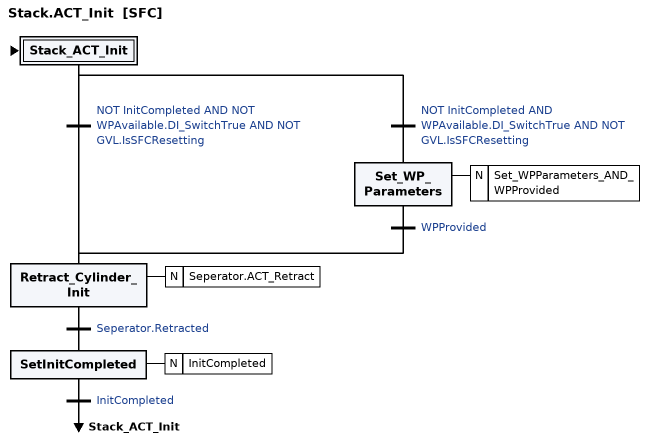
INITIAL_STEP Stack_ACT_Init:
END_STEP
TRANSITION FROM Stack_ACT_Init TO Retract_Cylinder_Init
  := NOT InitCompleted AND NOT WPAvailable.DI_SwitchTrue AND NOT
                                                    GVL.IsSFCResetting;
END_TRANSITION
TRANSITION FROM Stack_ACT_Init TO Set_WP_Parameters
  := NOT InitCompleted AND WPAvailable.DI_SwitchTrue AND NOT
                                                    GVL.IsSFCResetting;
END_TRANSITION
STEP Set_WP_Parameters:
  Set_WPParameters_AND_WPProvided(N);
END_STEP
TRANSITION FROM Set_WP_Parameters TO Retract_Cylinder_Init
  := WPProvided;
END_TRANSITION
STEP Retract_Cylinder_Init:
  Seperator.ACT_Retract(N);
END_STEP
TRANSITION FROM Retract_Cylinder_Init TO SetInitCompleted
  := Seperator.Retracted;
END_TRANSITION
STEP SetInitCompleted:
  InitCompleted(N);
END_STEP
TRANSITION FROM SetInitCompleted TO Stack_ACT_Init
  := InitCompleted;
END_TRANSITION
END_ACTION
END_FUNCTION_BLOCK

FUNCTION_BLOCK Stamp
                                            VAR_INPUT
                                            //Hardware
                                            Panel : OperationPanel;
                                            PressureSensor : PressureSensor;
                                            PropValve : ProportionalValve;
                                            WPAvailable : MicroSwitch;
                                            StampingCylinder : MonostableCylinder;
                                            SlidingCylinder : BistableCylinder;

                                            //Software
                                            StartButton : BOOL;
                                            InitCompleted : BOOL;
                                            AutomaticExecuteCompleted : BOOL;
                                            EmergencyStop : BOOL;
                                            SoftwareEmergency : BOOL;
                                            EmergencyHandled : BOOL;
                                            SFCReset : BOOL; //Only for SFC implementation
                                            END_VAR
                                            VAR_OUTPUT
                                            //Software
                                            IsStamping : BOOL;
                                            WPStamped : BOOL;
                                            WPType_White : BOOL;
                                            WPType_Black : BOOL;
                                            WPType_Metallic : BOOL;
                                            END_VAR
                                            VAR
                                            //Software
                                            Timer : TON;
                                            Check_Allowed_To_Operate : BOOL;
                                            Check_WPType_White : BOOL;
                                            Check_WPType_Black : BOOL;
                                            Check_WPType_Metallic : BOOL;
                                            Check_Stamp_WPAvailable : BOOL;
                                            END_VAR

                                    Panel();
                                        StartButton := Panel.StartButton;
                                        EmergencyStop := Panel.EmergencyStop;
                                        Check_Allowed_To_Operate := Main.Crane_Allow_Stamp_to_Operate;
                                        Check_WPType_White:=Main.Crane_WPType_White;
                                        Check_WPType_Black:=Main.Crane_WPType_Black;
                                        Check_WPType_Metallic:=Main.Crane_WPType_Metallic;
                                        Check_Stamp_WPAvailable:=Main.Stamp_WPAvailable;
                                    
                                

ACTION ExtendStampingCylinder_AND_Timer1500ms:
                                            StampingCylinder.ACT_Extend();
                                                Timer(IN:=TRUE, PT:=T#1500MS);
                                            
                                        
END_ACTION

ACTION Reset_Pressure:
                                            PropValve.AO_SetPressure:=0;
                                            
                                        
END_ACTION

ACTION Reset_Timer:
                                            Timer(IN:=FALSE);
                                        
END_ACTION

ACTION Reset_Variables:
                                            InitCompleted := FALSE;
                                                AutomaticExecuteCompleted := FALSE;

                                                propValve.AO_SetPressure:=0;
                                                IsStamping:=FALSE;
                                                WPStamped:=FALSE;
                                                WPType_Black := FALSE;
                                                WPType_White := FALSE;
                                                WPType_Metallic := FALSE;
                                            
                                        
END_ACTION

ACTION Set_HeavyPressure:
                                            
                                                PropValve.AO_SetPressure:=7000;
                                            
                                        
END_ACTION

ACTION Set_LightPressure:
                                            
                                                PropValve.AO_SetPressure:=4000;
                                            
                                        
END_ACTION

ACTION Set_Timer1000ms:
                                            Timer(IN:=TRUE, PT:=T#1000MS);
                                            
                                        
END_ACTION

ACTION Set_Timer500ms:
                                            Timer(IN:=TRUE, PT:=T#500ms);
                                            
                                        
END_ACTION

ACTION Set_WPType:
                                            WPType_White :=
                                                Check_WPType_White;
                                                WPType_Black := Check_WPType_Black;
                                                WPType_Metallic := Check_WPType_Metallic;
                                            
                                        
END_ACTION

ACTION ACT_Stamp:
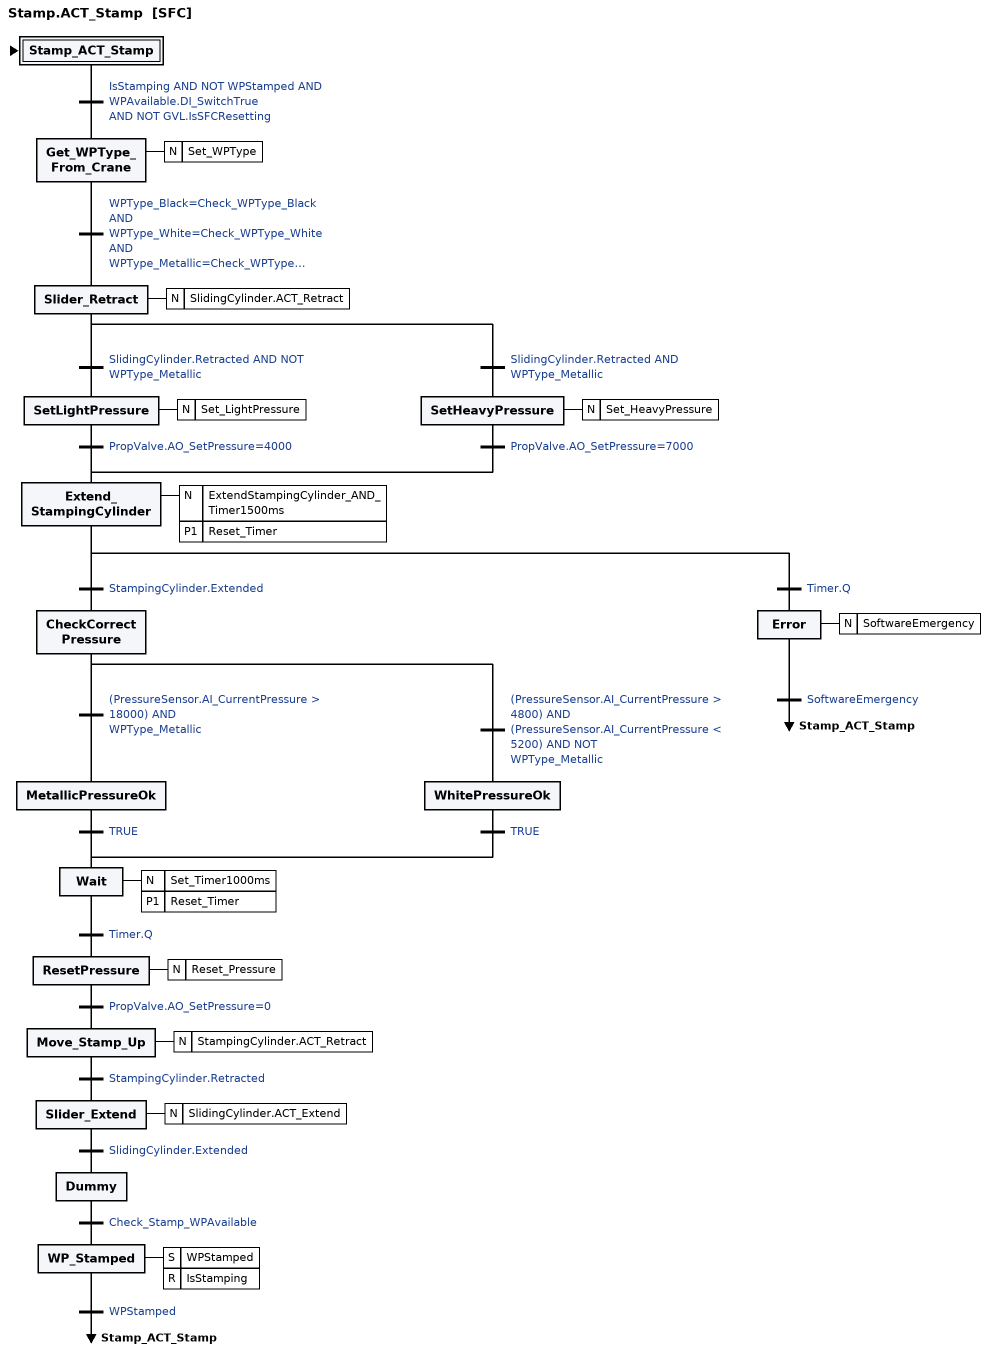
INITIAL_STEP Stamp_ACT_Stamp:
END_STEP
TRANSITION FROM Stamp_ACT_Stamp TO Get_WPType_From_Crane
  := IsStamping AND NOT WPStamped AND WPAvailable.DI_SwitchTrue
                                                    AND NOT GVL.IsSFCResetting;
END_TRANSITION
STEP Get_WPType_From_Crane:
  Set_WPType(N);
END_STEP
TRANSITION FROM Get_WPType_From_Crane TO Slider_Retract
  := WPType_Black=Check_WPType_Black AND
                                                    WPType_White=Check_WPType_White AND
                                                    WPType_Metallic=Check_WPType_Metallic;
END_TRANSITION
STEP Slider_Retract:
  SlidingCylinder.ACT_Retract(N);
END_STEP
TRANSITION FROM Slider_Retract TO SetLightPressure
  := SlidingCylinder.Retracted AND NOT WPType_Metallic;
END_TRANSITION
TRANSITION FROM Slider_Retract TO SetHeavyPressure
  := SlidingCylinder.Retracted AND WPType_Metallic;
END_TRANSITION
STEP SetLightPressure:
  Set_LightPressure(N);
END_STEP
TRANSITION FROM SetLightPressure TO Extend_StampingCylinder
  := PropValve.AO_SetPressure=4000;
END_TRANSITION
STEP SetHeavyPressure:
  Set_HeavyPressure(N);
END_STEP
TRANSITION FROM SetHeavyPressure TO Extend_StampingCylinder
  := PropValve.AO_SetPressure=7000;
END_TRANSITION
STEP Extend_StampingCylinder:
  ExtendStampingCylinder_AND_Timer1500ms(N);
  Reset_Timer(P1);
END_STEP
TRANSITION FROM Extend_StampingCylinder TO CheckCorrectPressure
  := StampingCylinder.Extended;
END_TRANSITION
TRANSITION FROM Extend_StampingCylinder TO Error
  := Timer.Q;
END_TRANSITION
STEP CheckCorrectPressure:
END_STEP
TRANSITION FROM CheckCorrectPressure TO MetallicPressureOk
  := (PressureSensor.AI_CurrentPressure > 18000) AND
                                                    WPType_Metallic;
END_TRANSITION
TRANSITION FROM CheckCorrectPressure TO WhitePressureOk
  := (PressureSensor.AI_CurrentPressure > 4800) AND
                                                    (PressureSensor.AI_CurrentPressure < 5200) AND NOT
                                                    WPType_Metallic;
END_TRANSITION
STEP MetallicPressureOk:
END_STEP
TRANSITION FROM MetallicPressureOk TO Wait
  := TRUE;
END_TRANSITION
STEP WhitePressureOk:
END_STEP
TRANSITION FROM WhitePressureOk TO Wait
  := TRUE;
END_TRANSITION
STEP Error:
  SoftwareEmergency(N);
END_STEP
TRANSITION FROM Error TO Stamp_ACT_Stamp
  := SoftwareEmergency;
END_TRANSITION
STEP Wait:
  Set_Timer1000ms(N);
  Reset_Timer(P1);
END_STEP
TRANSITION FROM Wait TO ResetPressure
  := Timer.Q;
END_TRANSITION
STEP ResetPressure:
  Reset_Pressure(N);
END_STEP
TRANSITION FROM ResetPressure TO Move_Stamp_Up
  := PropValve.AO_SetPressure=0;
END_TRANSITION
STEP Move_Stamp_Up:
  StampingCylinder.ACT_Retract(N);
END_STEP
TRANSITION FROM Move_Stamp_Up TO Slider_Extend
  := StampingCylinder.Retracted;
END_TRANSITION
STEP Slider_Extend:
  SlidingCylinder.ACT_Extend(N);
END_STEP
TRANSITION FROM Slider_Extend TO Dummy
  := SlidingCylinder.Extended;
END_TRANSITION
STEP Dummy:
END_STEP
TRANSITION FROM Dummy TO WP_Stamped
  := Check_Stamp_WPAvailable;
END_TRANSITION
STEP WP_Stamped:
  WPStamped(S);
  IsStamping(R);
END_STEP
TRANSITION FROM WP_Stamped TO Stamp_ACT_Stamp
  := WPStamped;
END_TRANSITION
END_ACTION

ACTION ACT_AutomaticExecute:
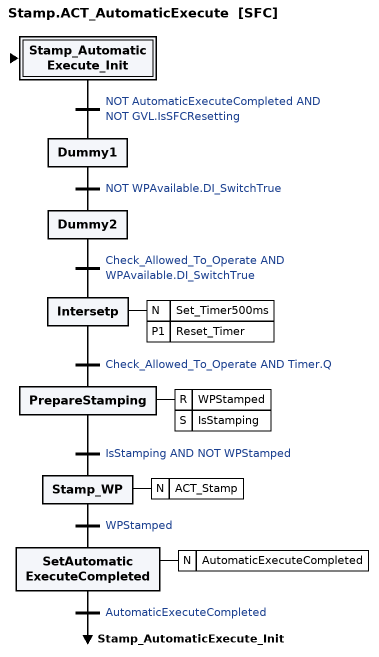
INITIAL_STEP Stamp_AutomaticExecute_Init:
END_STEP
TRANSITION FROM Stamp_AutomaticExecute_Init TO Dummy1
  := NOT AutomaticExecuteCompleted AND NOT GVL.IsSFCResetting;
END_TRANSITION
STEP Dummy1:
END_STEP
TRANSITION FROM Dummy1 TO Dummy2
  := NOT WPAvailable.DI_SwitchTrue;
END_TRANSITION
STEP Dummy2:
END_STEP
TRANSITION FROM Dummy2 TO Intersetp
  := Check_Allowed_To_Operate AND WPAvailable.DI_SwitchTrue;
END_TRANSITION
STEP Intersetp:
  Set_Timer500ms(N);
  Reset_Timer(P1);
END_STEP
TRANSITION FROM Intersetp TO PrepareStamping
  := Check_Allowed_To_Operate AND Timer.Q;
END_TRANSITION
STEP PrepareStamping:
  WPStamped(R);
  IsStamping(S);
END_STEP
TRANSITION FROM PrepareStamping TO Stamp_WP
  := IsStamping AND NOT WPStamped;
END_TRANSITION
STEP Stamp_WP:
  ACT_Stamp(N);
END_STEP
TRANSITION FROM Stamp_WP TO SetAutomaticExecuteCompleted
  := WPStamped;
END_TRANSITION
STEP SetAutomaticExecuteCompleted:
  AutomaticExecuteCompleted(N);
END_STEP
TRANSITION FROM SetAutomaticExecuteCompleted TO Stamp_AutomaticExecute_Init
  := AutomaticExecuteCompleted;
END_TRANSITION
END_ACTION

ACTION ACT_EmergencyStop:
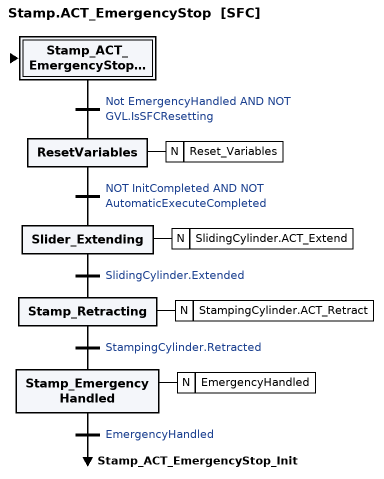
INITIAL_STEP Stamp_ACT_EmergencyStop_Init:
END_STEP
TRANSITION FROM Stamp_ACT_EmergencyStop_Init TO ResetVariables
  := Not EmergencyHandled AND NOT GVL.IsSFCResetting;
END_TRANSITION
STEP ResetVariables:
  Reset_Variables(N);
END_STEP
TRANSITION FROM ResetVariables TO Slider_Extending
  := NOT InitCompleted AND NOT AutomaticExecuteCompleted;
END_TRANSITION
STEP Slider_Extending:
  SlidingCylinder.ACT_Extend(N);
END_STEP
TRANSITION FROM Slider_Extending TO Stamp_Retracting
  := SlidingCylinder.Extended;
END_TRANSITION
STEP Stamp_Retracting:
  StampingCylinder.ACT_Retract(N);
END_STEP
TRANSITION FROM Stamp_Retracting TO Stamp_EmergencyHandled
  := StampingCylinder.Retracted;
END_TRANSITION
STEP Stamp_EmergencyHandled:
  EmergencyHandled(N);
END_STEP
TRANSITION FROM Stamp_EmergencyHandled TO Stamp_ACT_EmergencyStop_Init
  := EmergencyHandled;
END_TRANSITION
END_ACTION

ACTION ACT_Init:
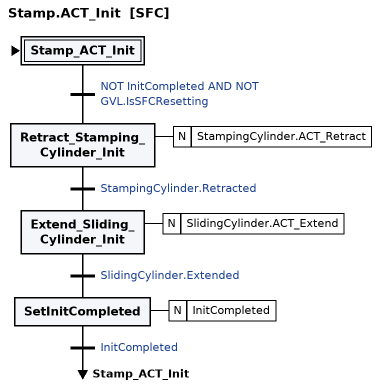
INITIAL_STEP Stamp_ACT_Init:
END_STEP
TRANSITION FROM Stamp_ACT_Init TO Retract_Stamping_Cylinder_Init
  := NOT InitCompleted AND NOT GVL.IsSFCResetting;
END_TRANSITION
STEP Retract_Stamping_Cylinder_Init:
  StampingCylinder.ACT_Retract(N);
END_STEP
TRANSITION FROM Retract_Stamping_Cylinder_Init TO Extend_Sliding_Cylinder_Init
  := StampingCylinder.Retracted;
END_TRANSITION
STEP Extend_Sliding_Cylinder_Init:
  SlidingCylinder.ACT_Extend(N);
END_STEP
TRANSITION FROM Extend_Sliding_Cylinder_Init TO SetInitCompleted
  := SlidingCylinder.Extended;
END_TRANSITION
STEP SetInitCompleted:
  InitCompleted(N);
END_STEP
TRANSITION FROM SetInitCompleted TO Stamp_ACT_Init
  := InitCompleted;
END_TRANSITION
END_ACTION
END_FUNCTION_BLOCK

FUNCTION_BLOCK PPU
                                            VAR_INPUT
                                            //Hardware
                                            Stack : Stack;
                                            Crane : Crane;
                                            LargeSortingConveyor : LargeSortingConveyor;
                                            Stamp : Stamp;
                                            //Software
                                            SFCReset : BOOL; //Only for SFC implementation
                                            END_VAR
                                            VAR_OUTPUT
                                            //Software
                                            StartButton : BOOL;
                                            InitCompleted : BOOL;
                                            AutomaticExecuteCompleted : BOOL;
                                            EmergencyStop : BOOL;
                                            EmergencyHandled : BOOL;
                                            SFCResetResetCompleted : BOOL; //Only for SFC implementation
                                            SFCResetCompleted : BOOL; //Only for SFC implementation
                                            END_VAR
                                            VAR
                                            END_VAR

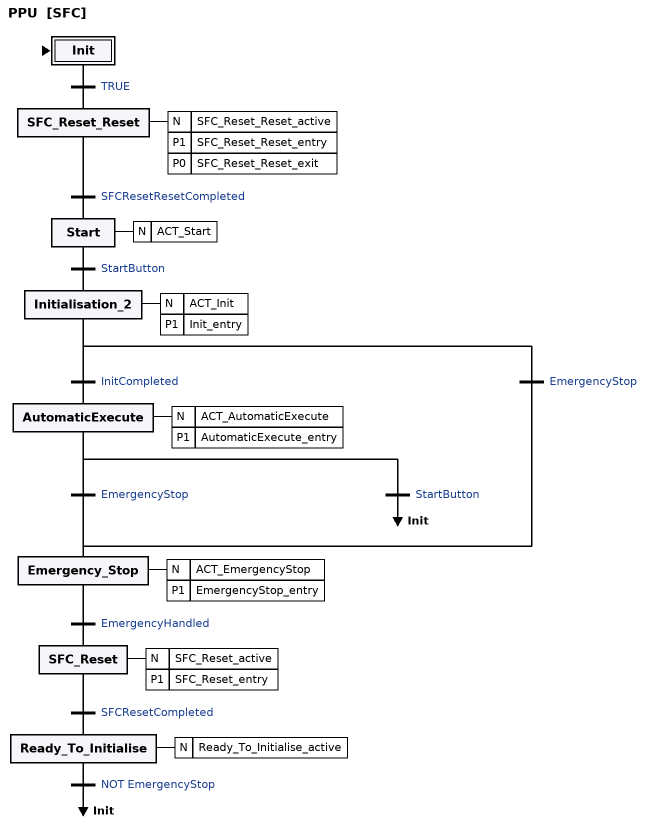
INITIAL_STEP Init:
END_STEP
TRANSITION FROM Init TO SFC_Reset_Reset
  := TRUE;
END_TRANSITION
STEP SFC_Reset_Reset:
  SFC_Reset_Reset_active(N);
  SFC_Reset_Reset_entry(P1);
  SFC_Reset_Reset_exit(P0);
END_STEP
TRANSITION FROM SFC_Reset_Reset TO Start
  := SFCResetResetCompleted;
END_TRANSITION
STEP Start:
  ACT_Start(N);
END_STEP
TRANSITION FROM Start TO Initialisation_2
  := StartButton;
END_TRANSITION
STEP Initialisation_2:
  ACT_Init(N);
  Init_entry(P1);
END_STEP
TRANSITION FROM Initialisation_2 TO AutomaticExecute
  := InitCompleted;
END_TRANSITION
TRANSITION FROM Initialisation_2 TO Emergency_Stop
  := EmergencyStop;
END_TRANSITION
STEP AutomaticExecute:
  ACT_AutomaticExecute(N);
  AutomaticExecute_entry(P1);
END_STEP
TRANSITION FROM AutomaticExecute TO Emergency_Stop
  := EmergencyStop;
END_TRANSITION
TRANSITION FROM AutomaticExecute TO Init
  := StartButton;
END_TRANSITION
STEP Emergency_Stop:
  ACT_EmergencyStop(N);
  EmergencyStop_entry(P1);
END_STEP
TRANSITION FROM Emergency_Stop TO SFC_Reset
  := EmergencyHandled;
END_TRANSITION
STEP SFC_Reset:
  SFC_Reset_active(N);
  SFC_Reset_entry(P1);
END_STEP
TRANSITION FROM SFC_Reset TO Ready_To_Initialise
  := SFCResetCompleted;
END_TRANSITION
STEP Ready_To_Initialise:
  Ready_To_Initialise_active(N);
END_STEP
TRANSITION FROM Ready_To_Initialise TO Init
  := NOT EmergencyStop;
END_TRANSITION

ACTION ACT_CheckEmergency:
                                            EmergencyStop :=
                                                Stack.EmergencyStop OR LargeSortingConveyor.EmergencyStop OR
                                                Stamp.EmergencyStop OR Crane.SoftwareEmergency OR
                                                Stamp.SoftwareEmergency;
                                            
                                        
END_ACTION

ACTION ACT_Start:
                                            StartButton := Stack.StartButton
                                                OR LargeSortingConveyor.StartButton OR Stamp.StartButton;
                                            
                                        
END_ACTION

ACTION AutomaticExecute_entry:
                                            
                                                AutomaticExecuteCompleted:=FALSE;

                                                LargeSortingConveyor.Panel.ACT_TurnLampWhite_Off();
                                                Stack.Panel.ACT_TurnLampWhite_Off();
                                                Stamp.Panel.ACT_TurnLampWhite_Off();
                                                LargeSortingConveyor.Panel.ACT_TurnLampGreen_On();
                                                Stack.Panel.ACT_TurnLampGreen_On();
                                                Stamp.Panel.ACT_TurnLampGreen_On();
                                            
                                        
END_ACTION

ACTION CallAll_AutomationExecutes:
                                            EmergencyStop :=
                                                Stack.EmergencyStop OR LargeSortingConveyor.EmergencyStop OR
                                                Stamp.EmergencyStop OR Crane.SoftwareEmergency OR
                                                Stamp.SoftwareEmergency;
                                                StartButton := Stack.StartButton OR LargeSortingConveyor.StartButton OR
                                                Stamp.StartButton;
                                                Crane.ACT_AutomaticExecute();
                                                Stack.ACT_AutomaticExecute();
                                                Stamp.ACT_AutomaticExecute();
                                                LargeSortingConveyor.ACT_AutomaticExecute();
                                            
                                        
END_ACTION

ACTION EmergencyStop_entry:
                                            EmergencyHandled:=FALSE;

                                                LargeSortingConveyor.Panel.ACT_TurnLampWhite_Off();
                                                Stack.Panel.ACT_TurnLampWhite_Off();
                                                Stamp.Panel.ACT_TurnLampWhite_Off();
                                                LargeSortingConveyor.Panel.ACT_TurnLampGreen_Off();
                                                Stack.Panel.ACT_TurnLampGreen_Off();
                                                Stamp.Panel.ACT_TurnLampGreen_Off();
                                            
                                        
END_ACTION

ACTION Init_entry:
                                            InitCompleted:=FALSE;

                                                LargeSortingConveyor.Panel.ACT_TurnLampWhite_On();
                                                Stack.Panel.ACT_TurnLampWhite_On();
                                                Stamp.Panel.ACT_TurnLampWhite_On();
                                                LargeSortingConveyor.Panel.ACT_TurnLampGreen_Off();
                                                Stack.Panel.ACT_TurnLampGreen_Off();
                                                Stamp.Panel.ACT_TurnLampGreen_Off();
                                            
                                        
END_ACTION

ACTION Ready_To_Initialise_active:
                                            EmergencyStop :=
                                                Stack.EmergencyStop OR LargeSortingConveyor.EmergencyStop OR
                                                Stamp.EmergencyStop OR Crane.SoftwareEmergency OR
                                                Stamp.SoftwareEmergency;
                                                StartButton := Stack.StartButton OR LargeSortingConveyor.StartButton OR
                                                Stamp.StartButton;
                                                IF(StartButton)THEN
                                                Stamp.SoftwareEmergency:=FALSE;
                                                Crane.SoftwareEmergency:=FALSE;
                                                END_IF
                                            
                                        
END_ACTION

ACTION SFC_Reset_active:
                                            (*PPU*)
                                                //Variables
                                                InitCompleted:=FALSE;
                                                AutomaticExecuteCompleted:=FALSE;

                                                (*Crane Reset*)
                                                Crane(SFCReset:=TRUE);
                                                Crane.ACT_Init(SFCReset:=TRUE);
                                                Crane.ACT_AutomaticExecute(SFCReset:=TRUE);
                                                Crane.ACT_EmergencyStop(SFCReset:=TRUE);
                                                Crane.ACT_MoveToConveyor(SFCReset:=TRUE);
                                                Crane.ACT_MoveToStack(SFCReset:=TRUE);
                                                Crane.ACT_MoveToStamp(SFCReset:=TRUE);
                                                Crane.ACT_PickUpWP(SFCReset:=TRUE);
                                                Crane.ACT_PutDownWP(SFCReset:=TRUE);

                                                (*LargeSortingConveyor Reset*)
                                                LargeSortingConveyor(SFCReset:=TRUE);
                                                LargeSortingConveyor.ACT_Init(SFCReset:=TRUE);
                                                LargeSortingConveyor.ACT_AutomaticExecute(SFCReset:=TRUE);
                                                LargeSortingConveyor.ACT_ChangeTarget(SFCReset:=TRUE);
                                                LargeSortingConveyor.ACT_CheckWPType(SFCReset:=TRUE);
                                                LargeSortingConveyor.ACT_SortWP(SFCReset:=TRUE);

                                                (*Stack Reset*)
                                                Stack(SFCReset:=TRUE);
                                                Stack.ACT_Init(SFCReset:=TRUE);
                                                Stack.ACT_AutomaticExecute(SFCReset:=TRUE);
                                                Stack.ACT_ProvideWP(SFCReset:=TRUE);

                                                (*Stamp Reset*)
                                                Stamp(SFCReset:=TRUE);
                                                Stamp.ACT_Init(SFCReset:=TRUE);
                                                Stamp.ACT_AutomaticExecute(SFCReset:=TRUE);
                                                Stamp.ACT_Stamp(SFCReset:=TRUE);

                                                SFCResetCompleted:=TRUE;
                                            
                                        
END_ACTION

ACTION SFC_Reset_entry:
                                            SFCResetCompleted:=FALSE;
                                                GVL.IsSFCResetting:=TRUE;
                                            
                                        
END_ACTION

ACTION SFC_Reset_Reset_active:
                                            (*Crane Reset*)
                                                Crane(SFCReset:=FALSE);
                                                Crane.ACT_Init(SFCReset:=FALSE);
                                                Crane.ACT_AutomaticExecute(SFCReset:=FALSE);
                                                Crane.ACT_EmergencyStop(SFCReset:=FALSE);
                                                Crane.ACT_MoveToConveyor(SFCReset:=FALSE);
                                                Crane.ACT_MoveToStack(SFCReset:=FALSE);
                                                Crane.ACT_MoveToStamp(SFCReset:=FALSE);
                                                Crane.ACT_PickUpWP(SFCReset:=FALSE);
                                                Crane.ACT_PutDownWP(SFCReset:=FALSE);
                                                Crane.LiftingCylinder.ACT_Retract();
                                                Crane.Gripper.ACT_Release();
                                                Crane.Table.Motor.ACT_Stop();
                                                //Variables
                                                Crane.InitCompleted:=FALSE;
                                                Crane.AutomaticExecuteCompleted:=FALSE;
                                                Crane.Conveyor_AllowedToOperate:=FALSE;
                                                Crane.Stamp_AllowedToOperate:=FALSE;
                                                Crane.SoftwareEmergency:=FALSE;
                                                Crane.EmergencyHandled:=FALSE;
                                                Crane.SFCReset:=FALSE;


                                                (*LargeSortingConveyor Reset*)
                                                LargeSortingConveyor(SFCReset:=FALSE);
                                                LargeSortingConveyor.ACT_Init(SFCReset:=FALSE);
                                                LargeSortingConveyor.ACT_AutomaticExecute(SFCReset:=FALSE);
                                                LargeSortingConveyor.ACT_ChangeTarget(SFCReset:=FALSE);
                                                LargeSortingConveyor.ACT_CheckWPType(SFCReset:=FALSE);
                                                LargeSortingConveyor.ACT_SortWP(SFCReset:=FALSE);
                                                LargeSortingConveyor.Motor.ACT_Stop();
                                                LargeSortingConveyor.Seperator1.ACT_Retract();
                                                LargeSortingConveyor.Seperator2.ACT_Retract();
                                                //Variables
                                                LargeSortingConveyor.SFCReset:=FALSE;

                                                (*Stack Reset*)
                                                Stack(SFCReset:=FALSE);
                                                Stack.ACT_Init(SFCReset:=FALSE);
                                                Stack.ACT_AutomaticExecute(SFCReset:=FALSE);
                                                Stack.ACT_ProvideWP(SFCReset:=FALSE);
                                                Stack.Seperator.ACT_Retract();
                                                //Variables
                                                Stack.InitCompleted:=FALSE;
                                                Stack.AutomaticExecuteCompleted:=FALSE;
                                                Stack.EmergencyHandled:=FALSE;
                                                Stack.SFCReset:=FALSE;

                                                (*Stamp Reset*)
                                                Stamp(SFCReset:=FALSE);
                                                Stamp.ACT_Init(SFCReset:=FALSE);
                                                Stamp.ACT_AutomaticExecute(SFCReset:=FALSE);
                                                Stamp.ACT_Stamp(SFCReset:=FALSE);
                                                Stamp.StampingCylinder.ACT_Retract();
                                                Stamp.SlidingCylinder.ACT_Extend();
                                                //Variables
                                                Stamp.InitCompleted:=FALSE;
                                                Stamp.AutomaticExecuteCompleted:=FALSE;
                                                Stamp.EmergencyHandled:=FALSE;
                                                Stamp.SFCReset:=FALSE;

                                                SFCResetResetCompleted:=TRUE;
                                                SFCResetCompleted:=TRUE;
                                            
                                        
END_ACTION

ACTION SFC_Reset_Reset_entry:
                                            SFCResetResetCompleted:=FALSE;
                                                GVL.IsSFCResetting:=TRUE;
                                            
                                        
END_ACTION

ACTION SFC_Reset_Reset_exit:
                                            GVL.IsSFCResetting:=FALSE;
                                            
                                        
END_ACTION

ACTION ACT_AutomaticExecute:
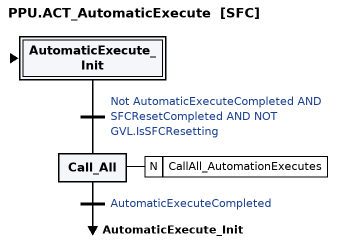
INITIAL_STEP AutomaticExecute_Init:
END_STEP
TRANSITION FROM AutomaticExecute_Init TO Call_All
  := Not AutomaticExecuteCompleted AND SFCResetCompleted AND NOT
                                                    GVL.IsSFCResetting;
END_TRANSITION
STEP Call_All:
  CallAll_AutomationExecutes(N);
END_STEP
TRANSITION FROM Call_All TO AutomaticExecute_Init
  := AutomaticExecuteCompleted;
END_TRANSITION
END_ACTION

ACTION ACT_EmergencyStop:
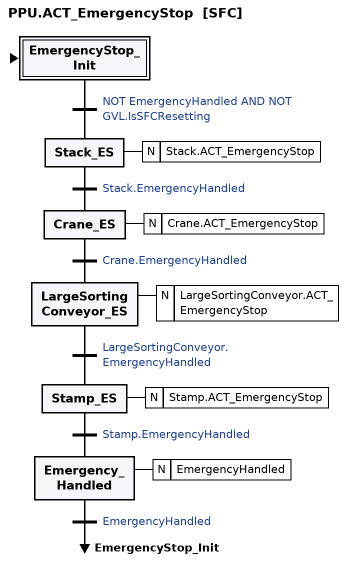
INITIAL_STEP EmergencyStop_Init:
END_STEP
TRANSITION FROM EmergencyStop_Init TO Stack_ES
  := NOT EmergencyHandled AND NOT GVL.IsSFCResetting;
END_TRANSITION
STEP Stack_ES:
  Stack.ACT_EmergencyStop(N);
END_STEP
TRANSITION FROM Stack_ES TO Crane_ES
  := Stack.EmergencyHandled;
END_TRANSITION
STEP Crane_ES:
  Crane.ACT_EmergencyStop(N);
END_STEP
TRANSITION FROM Crane_ES TO LargeSortingConveyor_ES
  := Crane.EmergencyHandled;
END_TRANSITION
STEP LargeSortingConveyor_ES:
  LargeSortingConveyor.ACT_EmergencyStop(N);
END_STEP
TRANSITION FROM LargeSortingConveyor_ES TO Stamp_ES
  := LargeSortingConveyor.EmergencyHandled;
END_TRANSITION
STEP Stamp_ES:
  Stamp.ACT_EmergencyStop(N);
END_STEP
TRANSITION FROM Stamp_ES TO Emergency_Handled
  := Stamp.EmergencyHandled;
END_TRANSITION
STEP Emergency_Handled:
  EmergencyHandled(N);
END_STEP
TRANSITION FROM Emergency_Handled TO EmergencyStop_Init
  := EmergencyHandled;
END_TRANSITION
END_ACTION

ACTION ACT_Init:
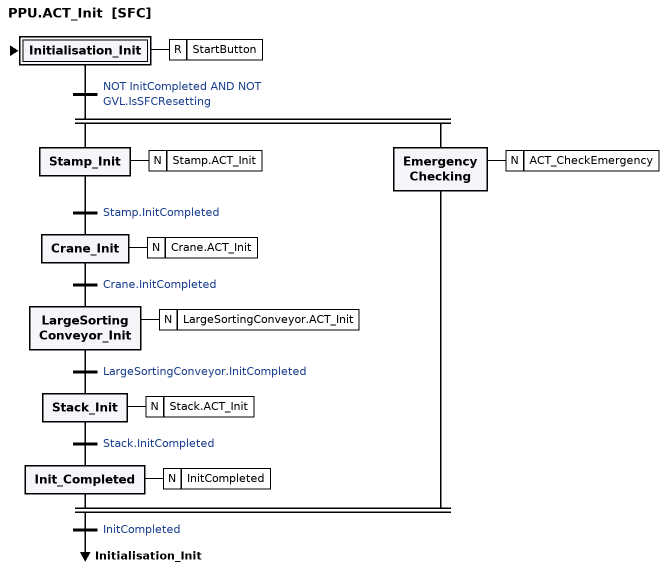
INITIAL_STEP Initialisation_Init:
  StartButton(R);
END_STEP
TRANSITION FROM Initialisation_Init TO (Stamp_Init, EmergencyChecking)
  := NOT InitCompleted AND NOT GVL.IsSFCResetting;
END_TRANSITION
STEP Stamp_Init:
  Stamp.ACT_Init(N);
END_STEP
TRANSITION FROM Stamp_Init TO Crane_Init
  := Stamp.InitCompleted;
END_TRANSITION
STEP Crane_Init:
  Crane.ACT_Init(N);
END_STEP
TRANSITION FROM Crane_Init TO LargeSortingConveyor_Init
  := Crane.InitCompleted;
END_TRANSITION
STEP LargeSortingConveyor_Init:
  LargeSortingConveyor.ACT_Init(N);
END_STEP
TRANSITION FROM LargeSortingConveyor_Init TO Stack_Init
  := LargeSortingConveyor.InitCompleted;
END_TRANSITION
STEP Stack_Init:
  Stack.ACT_Init(N);
END_STEP
TRANSITION FROM Stack_Init TO Init_Completed
  := Stack.InitCompleted;
END_TRANSITION
STEP Init_Completed:
  InitCompleted(N);
END_STEP
TRANSITION FROM (Init_Completed, EmergencyChecking) TO Initialisation_Init
  := InitCompleted;
END_TRANSITION
STEP EmergencyChecking:
  ACT_CheckEmergency(N);
END_STEP
END_ACTION
END_FUNCTION_BLOCK

CONFIGURATION Application
  RESOURCE Scenario_12 ON PLC
(* global variable list GVL *)
{attribute 'qualified_only'}
                                    VAR_GLOBAL
                                    IsSFCResetting : BOOL;
                                    END_VAR
    TASK PlcTask(INTERVAL := T#0ms, PRIORITY := 20);
    PROGRAM MAIN WITH PlcTask : MAIN;
  END_RESOURCE
END_CONFIGURATION
